FUNCTION_BLOCK FB_CartCheck
VAR_INPUT
END_VAR
VAR_OUTPUT
END_VAR
VAR
	// joint error flag
	m_jointErrFlag :ARRAY[1..4] OF BOOL:=[4(FALSE)];
	
	// joint control error flag
	m_jntCtrlErrFlag :vec4b;
	m_jntCtrlErrCounts :Vec4i;
	m_jntEncErr :Vec4d;
	
	// joint encoder error flag
	m_jntEncErrFlag :vec4b;
	m_jntEncErrCounts :Vec4i;
	m_jntCtrlErr : Vec4d;
	
	// joint velocity error flag
	m_jntVelErrFlag :vec4b;
	m_jntVelErrCounts  :Vec4i;
	
	// joint position limit error flag
	m_jntLimitErrFlag :Vec4b;
	m_jntLimitErrCounts :Vec4i;
	
END_VAR

METHOD check : BOOL
VAR_IN_OUT CONSTANT
	i_cartStatus : ST_CartStatus;
	i_cartJointData :ST_CartJointData;
END_VAR
VAR_OUTPUT
	o_errorFlag :ARRAY[1..4] OF BOOL ;
END_VAR

VAR
	i ,j:INT ;
END_VAR
// return if cart not init
IF NOT(i_cartStatus.m_initFlag) THEN
	RETURN;
END_IF

// joint control error
jntCtrlErrCheck(i_cartJointData.m_cmdJntPos, i_cartJointData.m_curJntPos);

// encoder error
jntEncErrCheck(i_cartJointData.m_curMotorPos, i_cartJointData.m_curLinkPos);

// joint velocity error
jntVelCheck(i_cartJointData.m_curJntVel);

// joint limit 
jntLimitCheck(i_cartJointData.m_curJntPos);
	
FOR i:=1 TO 4 DO 
	// stop check if arm is already in error state
	IF  m_jointErrFlag[i] THEN 
		CONTINUE;
	END_IF
	
	// final arm error status check
	IF m_jntCtrlErrFlag[i] OR  m_jntEncErrFlag[i] OR m_jntVelErrFlag[i] OR m_jntLimitErrFlag[i] THEN
		m_jointErrFlag[i]:=TRUE;
		EXIT;
	END_IF
	
END_FOR

o_errorFlag:=m_jointErrFlag;
END_METHOD

METHOD jntCtrlErrCheck : BOOL
VAR_INput
	i_cmdJntPos : Vec4d;
	i_curJntPos : Vec4d;
END_VAR

VAR
	i :INT;
END_VAR
// joint error check
FOR i:=1 TO 4 DO 
	// stop check if arm is already in error state
	IF m_jointErrFlag[i] THEN 
		CONTINUE;
	END_IF
	
	// error
	m_jntCtrlErr[i]:= i_cmdJntPos[i]-i_curJntPos[i];
	
	//check
	IF  ABS(m_jntCtrlErr[i]) > g_cartMaxJntCtrlErr[i] THEN
		m_jntCtrlErrCounts[i]:=m_jntCtrlErrCounts[i]+1;
	ELSE
		m_jntCtrlErrCounts[i] :=0;	
	END_IF
	m_jntCtrlErrFlag[i]:= m_jntCtrlErrCounts[i]>=g_faultTriggerCounts;
END_FOR
END_METHOD

METHOD jntEncErrCheck : BOOL
VAR_INput
	i_motorJntPos : Vec4d;
	i_linkJntPos : Vec4d;
END_VAR


VAR
	i :INT;
END_VAR
// joint error check
FOR i:=1 TO 4 DO 
	// stop check if arm is already in error state
	IF  m_jointErrFlag[i] THEN 
		CONTINUE;
	END_IF
	
	// error
	m_jntEncErr[i]:=i_motorJntPos[i]-i_linkJntPos[i];
	
	// check
	IF  ABS(m_jntEncErr[i]) > g_cartMaxJntEncErr[i] THEN
		m_jntEncErrCounts[i]:=m_jntEncErrCounts[i]+1;
	ELSE
		m_jntEncErrCounts[i] :=0;
	END_IF
	m_jntEncErrFlag[i]:= m_jntEncErrCounts[i]>=g_faultTriggerCounts;
END_FOR
END_METHOD

METHOD jntLimitCheck : bool
VAR_INPUT
	i_curJntPos : Vec4d;
END_VAR

VAR
	i:INT;
END_VAR
// joint position limit check
FOR i:=1 TO 4 DO 
	// stop check if arm is already in error state
	IF m_jointErrFlag[i] THEN 
		CONTINUE;
	END_IF
	
	// check
	IF  i_curJntPos[i] > GVL_CartJointParameters.g_maxJntPos[i] + g_cartJntPosLimitBuffer[i] OR
		i_curJntPos[i] < GVL_CartJointParameters.g_minJntPos[i] - g_cartJntPosLimitBuffer[i] THEN
		m_jntLimitErrCounts[i]:=m_jntLimitErrCounts[i]+1;
	ELSE
		m_jntLimitErrCounts[i] :=0;	
	END_IF
	m_jntLimitErrFlag[i]:= m_jntLimitErrCounts[i]>=g_faultTriggerCounts;
END_FOR
END_METHOD

METHOD jntVelCheck : bool
VAR_INPUT
	i_curJntVel : Vec4d;
END_VAR

VAR
	i:INT;
END_VAR
// joint velocity check
FOR i:=1 TO 4 DO 
	// stop check if arm is already in error state
	IF m_jointErrFlag[i] THEN 
		CONTINUE;
	END_IF
	
	// check
	IF  ABS(i_curJntVel[i]) > g_cartMaxJntVel[i] THEN
		m_jntVelErrCounts[i]:=m_jntVelErrCounts[i]+1;
	ELSE
		m_jntVelErrCounts[i] :=0;
	END_IF
	m_jntVelErrFlag[i]:= m_jntVelErrCounts[i]>=g_faultTriggerCounts;
END_FOR
END_METHOD

END_FUNCTION_BLOCK

(* stored: Version 1.1.0.1, ProductVersion 3.1.4024.12
   POU FB_CartCheck: Id {d1534ad2-2f8c-4055-becf-7fdf37e415fb}, SpecialFunc None
   Method check: Id {bef3b6ff-c9e8-4fbc-b2db-c79fe876dc97}
   Method jntCtrlErrCheck: Id {b4d4ba72-29e3-4420-ae1e-373c74cf8376}
   Method jntEncErrCheck: Id {01e25a9a-c621-44bd-8eb0-9ef81dee62f4}
   Method jntLimitCheck: Id {cd785ed3-1bd5-43af-9d92-dd40cbaa425b}
   Method jntVelCheck: Id {2e8b7dd4-14fe-4751-887c-4c0610d0cb5e} *)
